FUNCTION_BLOCK RT_E_EC_COUPLER (* Coupling two succeeding event chains *)
  (* Description: Copyright (c) 2008 ACIN This program and the accompanying materials are made available under the terms of the Eclipse Public License 2.0 which is available at https://www.eclipse.org/legal/epl-2.0/ SPDX-License-Identifier: EPL-2.0 *)
  (* Version 1.0, 2008-07-10, Alois Zoitl, ACIN *)
  (* Version 2.0, 2022-09-15, Michael Hansal, add WCET input *)
  (* Version 3.0, 2025-04-14, Patrick Aigner, changed package *)
  PACKAGE eclipse4diac::rtevents;
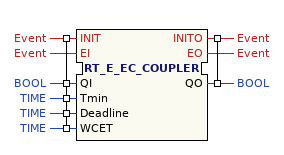
  EVENT_INPUT
    INIT WITH QI, Tmin, Deadline, WCET;
    EI; (* Event input *)
  END_EVENT
  EVENT_OUTPUT
    INITO WITH QO;
    EO; (* Event output *)
  END_EVENT
  VAR_INPUT
    QI : BOOL;
    Tmin : TIME;
    Deadline : TIME;
    WCET : TIME;
  END_VAR
  VAR_OUTPUT
    QO : BOOL;
  END_VAR
END_FUNCTION_BLOCK
